{attribute 'qualified_only'}
{attribute 'strict'}
{attribute 'to_string'}
TYPE E_LedColor :
(
    Off := 0,
    Red := 1,
    Green := 2,
    Blue := 3,
    Yellow := 4,
    Cyan := 5,
    Magenta := 6,
    White := 7
) USINT := Off;
END_TYPE

(* stored: Version 1.1.0.1, ProductVersion 3.1.4026.17
   DUT E_LedColor: Id {be9c6439-73b4-4aec-972b-87ca99f44a66} *)
